FUNCTION_BLOCK FB_CarrierReset
VAR_INPUT
	Execute : BOOL;
END_VAR
VAR_OUTPUT
	Busy	: BOOL;
	Done	: BOOL;
	Error	: BOOL;
END_VAR
VAR
	X_AxisReset	: MC_Reset;
	Z_AxisReset	: MC_Reset;

	{attribute 'hide'}
	_X_Axis :POINTER TO AXIS_REF;
	{attribute 'hide'}
	_Z_Axis :POINTER TO AXIS_REF;
	_SetPoint : ST_CarrierSetpoint;
END_VAR

IF _X_Axis= 0 OR _Z_Axis=0 THEN
	RETURN;
END_IF

X_AxisReset(Axis	:= _X_Axis^,
			Execute	:= Execute AND _X_Axis^.Status.Error);

Z_AxisReset(Axis	:= _Z_Axis^,
			Execute	:= Execute AND _Z_Axis^.Status.Error);

Busy := X_AxisReset.Busy OR Z_AxisReset.Busy;

Done := X_AxisReset.Done AND Z_AxisReset.Done;

Error := X_AxisReset.Error OR Z_AxisReset.Error;

PROPERTY X_AxisRef : POINTER TO AXIS_REF
GET
X_AxisRef := _X_Axis;
END_GET
SET
_X_Axis := X_AxisRef;
END_SET
END_PROPERTY

PROPERTY Z_AxisRef : POINTER TO AXIS_REF
GET
Z_AxisRef := _Z_Axis;
END_GET
SET
_Z_Axis := Z_AxisRef;
END_SET
END_PROPERTY

END_FUNCTION_BLOCK

(* stored: Version 1.1.0.1, ProductVersion 3.1.4024.12
   POU FB_CarrierReset: Id {b990260e-59ae-4992-829e-5901fb48bceb}, SpecialFunc None
   Property X_AxisRef: Id {5260bef5-2298-491f-9725-d71827cc0783}
   Get Get: Id {03705336-211d-47b3-95b3-f50a7847fcca}
   Set Set: Id {e75de4b7-6ea7-4e0d-b645-c0bd19391d59}
   Property Z_AxisRef: Id {33f0f1c7-28a6-4dfb-937a-97c2b92458c6}
   Get Get: Id {ef67b652-e2a5-4887-835e-f1ad55ca1908}
   Set Set: Id {e9a15d2d-4b28-4db3-bbbf-404f13d01f18} *)
